// TIA Portal V20 export
TYPE "LBP_typeTMSpindleMT"
TITLE = Tool management / Gestion des outils
// User data type for block LBP_TMSpindleMT [DB1072] / Type de données utilisateur pour bloc LBP_TMSpindleMT [DB1072]
   STRUCT
      MTIF : Array[1..16] of Struct
         DistanceCoding : Int;   // Type of distance coding ($TC_MTP_KD) / Type de codage de distance ($TC_MTP_KD)
         Places : Int;   // Number of locations of the multitool / Nombre d'emplacements Multitool
         Distance : Real;   // Multitool location distance / Distance de l'emplacement Multitool
         NewMTNo : Int;   // MT number of new tool / Numéro MT du nouvel outil
         NewPlace : Int;   // Multitool place number / Numéro d'emplacement Multitool
         OldMTNo : Int;   // MT number of previous tool / Numéro MT de l'outil précédent
         OldPlace : Int;   // Multitool place number / Numéro d'emplacement Multitool
         LocType : Int;   // Tool new: location type / Nouvel outil : type d'emplacement
         SLeft : Int;   // Tool new: size left / Nouvel outil : taille côté gauche
         SRight : Int;   // Tool new: size right / Nouvel outil : taille côté droit
         STop : Int;   // Tool new: size top / Nouvel outil : taille dessus
         SBottom : Int;   // Tool new: size bottom / Nouvel outil : taille dessous
         TInBuffer : Bool;   // ID for tools in buffer / ID pour outils dans tampon
         IgnoreDisabled : Bool;   // Ignore disabled / Ignorer désactivation
         Unload : Bool;   // To be unloaded / À décharger
         Load : Bool;   // To be loaded / À charger
         MasterTool : Bool;   // Tool is the master tool / L'outil est un outil principal
         n26_5 : Bool;   // Reserved / Réservé
         n26_6 : Bool;   // Reserved / Réservé
         HandTool : Bool;   // Hand tool / Outil manuel
         Active : Bool;   // Active tool / Outil actif
         Enabled : Bool;   // Tool enabled / Outil activé
         Disabled : Bool;   // Tool disabled / Outil désactivé
         Measured : Bool;   // Tool measured / Outil mesuré
         Prewarn : Bool;   // Prewarning limit reached / Seuil de préavis atteint
         Change : Bool;   // Tool being changed / Outil en cours de changement
         FixedLoc : Bool;   // Tool fixed location coded / Emplacement fixe d'outil codé
         Used : Bool;   // Tool was in use / Outil a été utilisé
         TNo : Int;   // Tool new: T number / Nouvel outil : numéro d'outil
         Toolholder : Int;   // Toolholder number as tool compensation reference / Numéro de porte-outil en tant que référence pour la compensation d'outil
         MyMag : Int;   // Multitool number the tool is loaded onto / Numéro Multitool dans lequel l'outil est chargé
         MyPlace : Int;   // Multitool place number / Numéro d'emplacement Multitool
         reserved : Array[1..7] of Int;   // Reserved / Réservé
      END_STRUCT;
   END_STRUCT;
   // // MTIF[2].DistanceCoding : Type of distance coding ($TC_MTP_KD) / Type de codage de distance ($TC_MTP_KD)
   // // MTIF[3].DistanceCoding : Type of distance coding ($TC_MTP_KD) / Type de codage de distance ($TC_MTP_KD)
   // // MTIF[4].DistanceCoding : Type of distance coding ($TC_MTP_KD) / Type de codage de distance ($TC_MTP_KD)
   // // MTIF[5].DistanceCoding : Type of distance coding ($TC_MTP_KD) / Type de codage de distance ($TC_MTP_KD)
   // // MTIF[6].DistanceCoding : Type of distance coding ($TC_MTP_KD) / Type de codage de distance ($TC_MTP_KD)
   // // MTIF[7].DistanceCoding : Type of distance coding ($TC_MTP_KD) / Type de codage de distance ($TC_MTP_KD)
   // // MTIF[8].DistanceCoding : Type of distance coding ($TC_MTP_KD) / Type de codage de distance ($TC_MTP_KD)
   // // MTIF[9].DistanceCoding : Type of distance coding ($TC_MTP_KD) / Type de codage de distance ($TC_MTP_KD)
   // // MTIF[10].DistanceCoding : Type of distance coding ($TC_MTP_KD) / Type de codage de distance ($TC_MTP_KD)
   // // MTIF[11].DistanceCoding : Type of distance coding ($TC_MTP_KD) / Type de codage de distance ($TC_MTP_KD)
   // // MTIF[12].DistanceCoding : Type of distance coding ($TC_MTP_KD) / Type de codage de distance ($TC_MTP_KD)
   // // MTIF[13].DistanceCoding : Type of distance coding ($TC_MTP_KD) / Type de codage de distance ($TC_MTP_KD)
   // // MTIF[14].DistanceCoding : Type of distance coding ($TC_MTP_KD) / Type de codage de distance ($TC_MTP_KD)
   // // MTIF[15].DistanceCoding : Type of distance coding ($TC_MTP_KD) / Type de codage de distance ($TC_MTP_KD)
   // // MTIF[16].DistanceCoding : Type of distance coding ($TC_MTP_KD) / Type de codage de distance ($TC_MTP_KD)
   // // MTIF[2].Places : Number of locations of the multitool / Nombre d'emplacements Multitool
   // // MTIF[3].Places : Number of locations of the multitool / Nombre d'emplacements Multitool
   // // MTIF[4].Places : Number of locations of the multitool / Nombre d'emplacements Multitool
   // // MTIF[5].Places : Number of locations of the multitool / Nombre d'emplacements Multitool
   // // MTIF[6].Places : Number of locations of the multitool / Nombre d'emplacements Multitool
   // // MTIF[7].Places : Number of locations of the multitool / Nombre d'emplacements Multitool
   // // MTIF[8].Places : Number of locations of the multitool / Nombre d'emplacements Multitool
   // // MTIF[9].Places : Number of locations of the multitool / Nombre d'emplacements Multitool
   // // MTIF[10].Places : Number of locations of the multitool / Nombre d'emplacements Multitool
   // // MTIF[11].Places : Number of locations of the multitool / Nombre d'emplacements Multitool
   // // MTIF[12].Places : Number of locations of the multitool / Nombre d'emplacements Multitool
   // // MTIF[13].Places : Number of locations of the multitool / Nombre d'emplacements Multitool
   // // MTIF[14].Places : Number of locations of the multitool / Nombre d'emplacements Multitool
   // // MTIF[15].Places : Number of locations of the multitool / Nombre d'emplacements Multitool
   // // MTIF[16].Places : Number of locations of the multitool / Nombre d'emplacements Multitool
   // // MTIF[2].Distance : Multitool location distance / Distance de l'emplacement Multitool
   // // MTIF[3].Distance : Multitool location distance / Distance de l'emplacement Multitool
   // // MTIF[4].Distance : Multitool location distance / Distance de l'emplacement Multitool
   // // MTIF[5].Distance : Multitool location distance / Distance de l'emplacement Multitool
   // // MTIF[6].Distance : Multitool location distance / Distance de l'emplacement Multitool
   // // MTIF[7].Distance : Multitool location distance / Distance de l'emplacement Multitool
   // // MTIF[8].Distance : Multitool location distance / Distance de l'emplacement Multitool
   // // MTIF[9].Distance : Multitool location distance / Distance de l'emplacement Multitool
   // // MTIF[10].Distance : Multitool location distance / Distance de l'emplacement Multitool
   // // MTIF[11].Distance : Multitool location distance / Distance de l'emplacement Multitool
   // // MTIF[12].Distance : Multitool location distance / Distance de l'emplacement Multitool
   // // MTIF[13].Distance : Multitool location distance / Distance de l'emplacement Multitool
   // // MTIF[14].Distance : Multitool location distance / Distance de l'emplacement Multitool
   // // MTIF[15].Distance : Multitool location distance / Distance de l'emplacement Multitool
   // // MTIF[16].Distance : Multitool location distance / Distance de l'emplacement Multitool
   // // MTIF[2].NewMTNo : MT number of new tool / Numéro MT du nouvel outil
   // // MTIF[3].NewMTNo : MT number of new tool / Numéro MT du nouvel outil
   // // MTIF[4].NewMTNo : MT number of new tool / Numéro MT du nouvel outil
   // // MTIF[5].NewMTNo : MT number of new tool / Numéro MT du nouvel outil
   // // MTIF[6].NewMTNo : MT number of new tool / Numéro MT du nouvel outil
   // // MTIF[7].NewMTNo : MT number of new tool / Numéro MT du nouvel outil
   // // MTIF[8].NewMTNo : MT number of new tool / Numéro MT du nouvel outil
   // // MTIF[9].NewMTNo : MT number of new tool / Numéro MT du nouvel outil
   // // MTIF[10].NewMTNo : MT number of new tool / Numéro MT du nouvel outil
   // // MTIF[11].NewMTNo : MT number of new tool / Numéro MT du nouvel outil
   // // MTIF[12].NewMTNo : MT number of new tool / Numéro MT du nouvel outil
   // // MTIF[13].NewMTNo : MT number of new tool / Numéro MT du nouvel outil
   // // MTIF[14].NewMTNo : MT number of new tool / Numéro MT du nouvel outil
   // // MTIF[15].NewMTNo : MT number of new tool / Numéro MT du nouvel outil
   // // MTIF[16].NewMTNo : MT number of new tool / Numéro MT du nouvel outil
   // // MTIF[2].NewPlace : Multitool place number / Numéro d'emplacement Multitool
   // // MTIF[3].NewPlace : Multitool place number / Numéro d'emplacement Multitool
   // // MTIF[4].NewPlace : Multitool place number / Numéro d'emplacement Multitool
   // // MTIF[5].NewPlace : Multitool place number / Numéro d'emplacement Multitool
   // // MTIF[6].NewPlace : Multitool place number / Numéro d'emplacement Multitool
   // // MTIF[7].NewPlace : Multitool place number / Numéro d'emplacement Multitool
   // // MTIF[8].NewPlace : Multitool place number / Numéro d'emplacement Multitool
   // // MTIF[9].NewPlace : Multitool place number / Numéro d'emplacement Multitool
   // // MTIF[10].NewPlace : Multitool place number / Numéro d'emplacement Multitool
   // // MTIF[11].NewPlace : Multitool place number / Numéro d'emplacement Multitool
   // // MTIF[12].NewPlace : Multitool place number / Numéro d'emplacement Multitool
   // // MTIF[13].NewPlace : Multitool place number / Numéro d'emplacement Multitool
   // // MTIF[14].NewPlace : Multitool place number / Numéro d'emplacement Multitool
   // // MTIF[15].NewPlace : Multitool place number / Numéro d'emplacement Multitool
   // // MTIF[16].NewPlace : Multitool place number / Numéro d'emplacement Multitool
   // // MTIF[2].OldMTNo : MT number of previous tool / Numéro MT de l'outil précédent
   // // MTIF[3].OldMTNo : MT number of previous tool / Numéro MT de l'outil précédent
   // // MTIF[4].OldMTNo : MT number of previous tool / Numéro MT de l'outil précédent
   // // MTIF[5].OldMTNo : MT number of previous tool / Numéro MT de l'outil précédent
   // // MTIF[6].OldMTNo : MT number of previous tool / Numéro MT de l'outil précédent
   // // MTIF[7].OldMTNo : MT number of previous tool / Numéro MT de l'outil précédent
   // // MTIF[8].OldMTNo : MT number of previous tool / Numéro MT de l'outil précédent
   // // MTIF[9].OldMTNo : MT number of previous tool / Numéro MT de l'outil précédent
   // // MTIF[10].OldMTNo : MT number of previous tool / Numéro MT de l'outil précédent
   // // MTIF[11].OldMTNo : MT number of previous tool / Numéro MT de l'outil précédent
   // // MTIF[12].OldMTNo : MT number of previous tool / Numéro MT de l'outil précédent
   // // MTIF[13].OldMTNo : MT number of previous tool / Numéro MT de l'outil précédent
   // // MTIF[14].OldMTNo : MT number of previous tool / Numéro MT de l'outil précédent
   // // MTIF[15].OldMTNo : MT number of previous tool / Numéro MT de l'outil précédent
   // // MTIF[16].OldMTNo : MT number of previous tool / Numéro MT de l'outil précédent
   // // MTIF[2].OldPlace : Multitool place number / Numéro d'emplacement Multitool
   // // MTIF[3].OldPlace : Multitool place number / Numéro d'emplacement Multitool
   // // MTIF[4].OldPlace : Multitool place number / Numéro d'emplacement Multitool
   // // MTIF[5].OldPlace : Multitool place number / Numéro d'emplacement Multitool
   // // MTIF[6].OldPlace : Multitool place number / Numéro d'emplacement Multitool
   // // MTIF[7].OldPlace : Multitool place number / Numéro d'emplacement Multitool
   // // MTIF[8].OldPlace : Multitool place number / Numéro d'emplacement Multitool
   // // MTIF[9].OldPlace : Multitool place number / Numéro d'emplacement Multitool
   // // MTIF[10].OldPlace : Multitool place number / Numéro d'emplacement Multitool
   // // MTIF[11].OldPlace : Multitool place number / Numéro d'emplacement Multitool
   // // MTIF[12].OldPlace : Multitool place number / Numéro d'emplacement Multitool
   // // MTIF[13].OldPlace : Multitool place number / Numéro d'emplacement Multitool
   // // MTIF[14].OldPlace : Multitool place number / Numéro d'emplacement Multitool
   // // MTIF[15].OldPlace : Multitool place number / Numéro d'emplacement Multitool
   // // MTIF[16].OldPlace : Multitool place number / Numéro d'emplacement Multitool
   // // MTIF[2].LocType : Tool new: location type / Nouvel outil : type d'emplacement
   // // MTIF[3].LocType : Tool new: location type / Nouvel outil : type d'emplacement
   // // MTIF[4].LocType : Tool new: location type / Nouvel outil : type d'emplacement
   // // MTIF[5].LocType : Tool new: location type / Nouvel outil : type d'emplacement
   // // MTIF[6].LocType : Tool new: location type / Nouvel outil : type d'emplacement
   // // MTIF[7].LocType : Tool new: location type / Nouvel outil : type d'emplacement
   // // MTIF[8].LocType : Tool new: location type / Nouvel outil : type d'emplacement
   // // MTIF[9].LocType : Tool new: location type / Nouvel outil : type d'emplacement
   // // MTIF[10].LocType : Tool new: location type / Nouvel outil : type d'emplacement
   // // MTIF[11].LocType : Tool new: location type / Nouvel outil : type d'emplacement
   // // MTIF[12].LocType : Tool new: location type / Nouvel outil : type d'emplacement
   // // MTIF[13].LocType : Tool new: location type / Nouvel outil : type d'emplacement
   // // MTIF[14].LocType : Tool new: location type / Nouvel outil : type d'emplacement
   // // MTIF[15].LocType : Tool new: location type / Nouvel outil : type d'emplacement
   // // MTIF[16].LocType : Tool new: location type / Nouvel outil : type d'emplacement
   // // MTIF[2].SLeft : Tool new: size left / Nouvel outil : taille côté gauche
   // // MTIF[3].SLeft : Tool new: size left / Nouvel outil : taille côté gauche
   // // MTIF[4].SLeft : Tool new: size left / Nouvel outil : taille côté gauche
   // // MTIF[5].SLeft : Tool new: size left / Nouvel outil : taille côté gauche
   // // MTIF[6].SLeft : Tool new: size left / Nouvel outil : taille côté gauche
   // // MTIF[7].SLeft : Tool new: size left / Nouvel outil : taille côté gauche
   // // MTIF[8].SLeft : Tool new: size left / Nouvel outil : taille côté gauche
   // // MTIF[9].SLeft : Tool new: size left / Nouvel outil : taille côté gauche
   // // MTIF[10].SLeft : Tool new: size left / Nouvel outil : taille côté gauche
   // // MTIF[11].SLeft : Tool new: size left / Nouvel outil : taille côté gauche
   // // MTIF[12].SLeft : Tool new: size left / Nouvel outil : taille côté gauche
   // // MTIF[13].SLeft : Tool new: size left / Nouvel outil : taille côté gauche
   // // MTIF[14].SLeft : Tool new: size left / Nouvel outil : taille côté gauche
   // // MTIF[15].SLeft : Tool new: size left / Nouvel outil : taille côté gauche
   // // MTIF[16].SLeft : Tool new: size left / Nouvel outil : taille côté gauche
   // // MTIF[2].SRight : Tool new: size right / Nouvel outil : taille côté droit
   // // MTIF[3].SRight : Tool new: size right / Nouvel outil : taille côté droit
   // // MTIF[4].SRight : Tool new: size right / Nouvel outil : taille côté droit
   // // MTIF[5].SRight : Tool new: size right / Nouvel outil : taille côté droit
   // // MTIF[6].SRight : Tool new: size right / Nouvel outil : taille côté droit
   // // MTIF[7].SRight : Tool new: size right / Nouvel outil : taille côté droit
   // // MTIF[8].SRight : Tool new: size right / Nouvel outil : taille côté droit
   // // MTIF[9].SRight : Tool new: size right / Nouvel outil : taille côté droit
   // // MTIF[10].SRight : Tool new: size right / Nouvel outil : taille côté droit
   // // MTIF[11].SRight : Tool new: size right / Nouvel outil : taille côté droit
   // // MTIF[12].SRight : Tool new: size right / Nouvel outil : taille côté droit
   // // MTIF[13].SRight : Tool new: size right / Nouvel outil : taille côté droit
   // // MTIF[14].SRight : Tool new: size right / Nouvel outil : taille côté droit
   // // MTIF[15].SRight : Tool new: size right / Nouvel outil : taille côté droit
   // // MTIF[16].SRight : Tool new: size right / Nouvel outil : taille côté droit
   // // MTIF[2].STop : Tool new: size top / Nouvel outil : taille dessus
   // // MTIF[3].STop : Tool new: size top / Nouvel outil : taille dessus
   // // MTIF[4].STop : Tool new: size top / Nouvel outil : taille dessus
   // // MTIF[5].STop : Tool new: size top / Nouvel outil : taille dessus
   // // MTIF[6].STop : Tool new: size top / Nouvel outil : taille dessus
   // // MTIF[7].STop : Tool new: size top / Nouvel outil : taille dessus
   // // MTIF[8].STop : Tool new: size top / Nouvel outil : taille dessus
   // // MTIF[9].STop : Tool new: size top / Nouvel outil : taille dessus
   // // MTIF[10].STop : Tool new: size top / Nouvel outil : taille dessus
   // // MTIF[11].STop : Tool new: size top / Nouvel outil : taille dessus
   // // MTIF[12].STop : Tool new: size top / Nouvel outil : taille dessus
   // // MTIF[13].STop : Tool new: size top / Nouvel outil : taille dessus
   // // MTIF[14].STop : Tool new: size top / Nouvel outil : taille dessus
   // // MTIF[15].STop : Tool new: size top / Nouvel outil : taille dessus
   // // MTIF[16].STop : Tool new: size top / Nouvel outil : taille dessus
   // // MTIF[2].SBottom : Tool new: size bottom / Nouvel outil : taille dessous
   // // MTIF[3].SBottom : Tool new: size bottom / Nouvel outil : taille dessous
   // // MTIF[4].SBottom : Tool new: size bottom / Nouvel outil : taille dessous
   // // MTIF[5].SBottom : Tool new: size bottom / Nouvel outil : taille dessous
   // // MTIF[6].SBottom : Tool new: size bottom / Nouvel outil : taille dessous
   // // MTIF[7].SBottom : Tool new: size bottom / Nouvel outil : taille dessous
   // // MTIF[8].SBottom : Tool new: size bottom / Nouvel outil : taille dessous
   // // MTIF[9].SBottom : Tool new: size bottom / Nouvel outil : taille dessous
   // // MTIF[10].SBottom : Tool new: size bottom / Nouvel outil : taille dessous
   // // MTIF[11].SBottom : Tool new: size bottom / Nouvel outil : taille dessous
   // // MTIF[12].SBottom : Tool new: size bottom / Nouvel outil : taille dessous
   // // MTIF[13].SBottom : Tool new: size bottom / Nouvel outil : taille dessous
   // // MTIF[14].SBottom : Tool new: size bottom / Nouvel outil : taille dessous
   // // MTIF[15].SBottom : Tool new: size bottom / Nouvel outil : taille dessous
   // // MTIF[16].SBottom : Tool new: size bottom / Nouvel outil : taille dessous
   // // MTIF[2].TInBuffer : ID for tools in buffer / ID pour outils dans tampon
   // // MTIF[3].TInBuffer : ID for tools in buffer / ID pour outils dans tampon
   // // MTIF[4].TInBuffer : ID for tools in buffer / ID pour outils dans tampon
   // // MTIF[5].TInBuffer : ID for tools in buffer / ID pour outils dans tampon
   // // MTIF[6].TInBuffer : ID for tools in buffer / ID pour outils dans tampon
   // // MTIF[7].TInBuffer : ID for tools in buffer / ID pour outils dans tampon
   // // MTIF[8].TInBuffer : ID for tools in buffer / ID pour outils dans tampon
   // // MTIF[9].TInBuffer : ID for tools in buffer / ID pour outils dans tampon
   // // MTIF[10].TInBuffer : ID for tools in buffer / ID pour outils dans tampon
   // // MTIF[11].TInBuffer : ID for tools in buffer / ID pour outils dans tampon
   // // MTIF[12].TInBuffer : ID for tools in buffer / ID pour outils dans tampon
   // // MTIF[13].TInBuffer : ID for tools in buffer / ID pour outils dans tampon
   // // MTIF[14].TInBuffer : ID for tools in buffer / ID pour outils dans tampon
   // // MTIF[15].TInBuffer : ID for tools in buffer / ID pour outils dans tampon
   // // MTIF[16].TInBuffer : ID for tools in buffer / ID pour outils dans tampon
   // // MTIF[2].IgnoreDisabled : Ignore disabled / Ignorer désactivation
   // // MTIF[3].IgnoreDisabled : Ignore disabled / Ignorer désactivation
   // // MTIF[4].IgnoreDisabled : Ignore disabled / Ignorer désactivation
   // // MTIF[5].IgnoreDisabled : Ignore disabled / Ignorer désactivation
   // // MTIF[6].IgnoreDisabled : Ignore disabled / Ignorer désactivation
   // // MTIF[7].IgnoreDisabled : Ignore disabled / Ignorer désactivation
   // // MTIF[8].IgnoreDisabled : Ignore disabled / Ignorer désactivation
   // // MTIF[9].IgnoreDisabled : Ignore disabled / Ignorer désactivation
   // // MTIF[10].IgnoreDisabled : Ignore disabled / Ignorer désactivation
   // // MTIF[11].IgnoreDisabled : Ignore disabled / Ignorer désactivation
   // // MTIF[12].IgnoreDisabled : Ignore disabled / Ignorer désactivation
   // // MTIF[13].IgnoreDisabled : Ignore disabled / Ignorer désactivation
   // // MTIF[14].IgnoreDisabled : Ignore disabled / Ignorer désactivation
   // // MTIF[15].IgnoreDisabled : Ignore disabled / Ignorer désactivation
   // // MTIF[16].IgnoreDisabled : Ignore disabled / Ignorer désactivation
   // // MTIF[2].Unload : To be unloaded / À décharger
   // // MTIF[3].Unload : To be unloaded / À décharger
   // // MTIF[4].Unload : To be unloaded / À décharger
   // // MTIF[5].Unload : To be unloaded / À décharger
   // // MTIF[6].Unload : To be unloaded / À décharger
   // // MTIF[7].Unload : To be unloaded / À décharger
   // // MTIF[8].Unload : To be unloaded / À décharger
   // // MTIF[9].Unload : To be unloaded / À décharger
   // // MTIF[10].Unload : To be unloaded / À décharger
   // // MTIF[11].Unload : To be unloaded / À décharger
   // // MTIF[12].Unload : To be unloaded / À décharger
   // // MTIF[13].Unload : To be unloaded / À décharger
   // // MTIF[14].Unload : To be unloaded / À décharger
   // // MTIF[15].Unload : To be unloaded / À décharger
   // // MTIF[16].Unload : To be unloaded / À décharger
   // // MTIF[2].Load : To be loaded / À charger
   // // MTIF[3].Load : To be loaded / À charger
   // // MTIF[4].Load : To be loaded / À charger
   // // MTIF[5].Load : To be loaded / À charger
   // // MTIF[6].Load : To be loaded / À charger
   // // MTIF[7].Load : To be loaded / À charger
   // // MTIF[8].Load : To be loaded / À charger
   // // MTIF[9].Load : To be loaded / À charger
   // // MTIF[10].Load : To be loaded / À charger
   // // MTIF[11].Load : To be loaded / À charger
   // // MTIF[12].Load : To be loaded / À charger
   // // MTIF[13].Load : To be loaded / À charger
   // // MTIF[14].Load : To be loaded / À charger
   // // MTIF[15].Load : To be loaded / À charger
   // // MTIF[16].Load : To be loaded / À charger
   // // MTIF[2].MasterTool : Tool is the master tool / L'outil est un outil principal
   // // MTIF[3].MasterTool : Tool is the master tool / L'outil est un outil principal
   // // MTIF[4].MasterTool : Tool is the master tool / L'outil est un outil principal
   // // MTIF[5].MasterTool : Tool is the master tool / L'outil est un outil principal
   // // MTIF[6].MasterTool : Tool is the master tool / L'outil est un outil principal
   // // MTIF[7].MasterTool : Tool is the master tool / L'outil est un outil principal
   // // MTIF[8].MasterTool : Tool is the master tool / L'outil est un outil principal
   // // MTIF[9].MasterTool : Tool is the master tool / L'outil est un outil principal
   // // MTIF[10].MasterTool : Tool is the master tool / L'outil est un outil principal
   // // MTIF[11].MasterTool : Tool is the master tool / L'outil est un outil principal
   // // MTIF[12].MasterTool : Tool is the master tool / L'outil est un outil principal
   // // MTIF[13].MasterTool : Tool is the master tool / L'outil est un outil principal
   // // MTIF[14].MasterTool : Tool is the master tool / L'outil est un outil principal
   // // MTIF[15].MasterTool : Tool is the master tool / L'outil est un outil principal
   // // MTIF[16].MasterTool : Tool is the master tool / L'outil est un outil principal
   // // MTIF[2].n26_5 : Reserved / Réservé
   // // MTIF[3].n26_5 : Reserved / Réservé
   // // MTIF[4].n26_5 : Reserved / Réservé
   // // MTIF[5].n26_5 : Reserved / Réservé
   // // MTIF[6].n26_5 : Reserved / Réservé
   // // MTIF[7].n26_5 : Reserved / Réservé
   // // MTIF[8].n26_5 : Reserved / Réservé
   // // MTIF[9].n26_5 : Reserved / Réservé
   // // MTIF[10].n26_5 : Reserved / Réservé
   // // MTIF[11].n26_5 : Reserved / Réservé
   // // MTIF[12].n26_5 : Reserved / Réservé
   // // MTIF[13].n26_5 : Reserved / Réservé
   // // MTIF[14].n26_5 : Reserved / Réservé
   // // MTIF[15].n26_5 : Reserved / Réservé
   // // MTIF[16].n26_5 : Reserved / Réservé
   // // MTIF[2].n26_6 : Reserved / Réservé
   // // MTIF[3].n26_6 : Reserved / Réservé
   // // MTIF[4].n26_6 : Reserved / Réservé
   // // MTIF[5].n26_6 : Reserved / Réservé
   // // MTIF[6].n26_6 : Reserved / Réservé
   // // MTIF[7].n26_6 : Reserved / Réservé
   // // MTIF[8].n26_6 : Reserved / Réservé
   // // MTIF[9].n26_6 : Reserved / Réservé
   // // MTIF[10].n26_6 : Reserved / Réservé
   // // MTIF[11].n26_6 : Reserved / Réservé
   // // MTIF[12].n26_6 : Reserved / Réservé
   // // MTIF[13].n26_6 : Reserved / Réservé
   // // MTIF[14].n26_6 : Reserved / Réservé
   // // MTIF[15].n26_6 : Reserved / Réservé
   // // MTIF[16].n26_6 : Reserved / Réservé
   // // MTIF[2].HandTool : Hand tool / Outil manuel
   // // MTIF[3].HandTool : Hand tool / Outil manuel
   // // MTIF[4].HandTool : Hand tool / Outil manuel
   // // MTIF[5].HandTool : Hand tool / Outil manuel
   // // MTIF[6].HandTool : Hand tool / Outil manuel
   // // MTIF[7].HandTool : Hand tool / Outil manuel
   // // MTIF[8].HandTool : Hand tool / Outil manuel
   // // MTIF[9].HandTool : Hand tool / Outil manuel
   // // MTIF[10].HandTool : Hand tool / Outil manuel
   // // MTIF[11].HandTool : Hand tool / Outil manuel
   // // MTIF[12].HandTool : Hand tool / Outil manuel
   // // MTIF[13].HandTool : Hand tool / Outil manuel
   // // MTIF[14].HandTool : Hand tool / Outil manuel
   // // MTIF[15].HandTool : Hand tool / Outil manuel
   // // MTIF[16].HandTool : Hand tool / Outil manuel
   // // MTIF[2].Active : Active tool / Outil actif
   // // MTIF[3].Active : Active tool / Outil actif
   // // MTIF[4].Active : Active tool / Outil actif
   // // MTIF[5].Active : Active tool / Outil actif
   // // MTIF[6].Active : Active tool / Outil actif
   // // MTIF[7].Active : Active tool / Outil actif
   // // MTIF[8].Active : Active tool / Outil actif
   // // MTIF[9].Active : Active tool / Outil actif
   // // MTIF[10].Active : Active tool / Outil actif
   // // MTIF[11].Active : Active tool / Outil actif
   // // MTIF[12].Active : Active tool / Outil actif
   // // MTIF[13].Active : Active tool / Outil actif
   // // MTIF[14].Active : Active tool / Outil actif
   // // MTIF[15].Active : Active tool / Outil actif
   // // MTIF[16].Active : Active tool / Outil actif
   // // MTIF[2].Enabled : Tool enabled / Outil activé
   // // MTIF[3].Enabled : Tool enabled / Outil activé
   // // MTIF[4].Enabled : Tool enabled / Outil activé
   // // MTIF[5].Enabled : Tool enabled / Outil activé
   // // MTIF[6].Enabled : Tool enabled / Outil activé
   // // MTIF[7].Enabled : Tool enabled / Outil activé
   // // MTIF[8].Enabled : Tool enabled / Outil activé
   // // MTIF[9].Enabled : Tool enabled / Outil activé
   // // MTIF[10].Enabled : Tool enabled / Outil activé
   // // MTIF[11].Enabled : Tool enabled / Outil activé
   // // MTIF[12].Enabled : Tool enabled / Outil activé
   // // MTIF[13].Enabled : Tool enabled / Outil activé
   // // MTIF[14].Enabled : Tool enabled / Outil activé
   // // MTIF[15].Enabled : Tool enabled / Outil activé
   // // MTIF[16].Enabled : Tool enabled / Outil activé
   // // MTIF[2].Disabled : Tool disabled / Outil désactivé
   // // MTIF[3].Disabled : Tool disabled / Outil désactivé
   // // MTIF[4].Disabled : Tool disabled / Outil désactivé
   // // MTIF[5].Disabled : Tool disabled / Outil désactivé
   // // MTIF[6].Disabled : Tool disabled / Outil désactivé
   // // MTIF[7].Disabled : Tool disabled / Outil désactivé
   // // MTIF[8].Disabled : Tool disabled / Outil désactivé
   // // MTIF[9].Disabled : Tool disabled / Outil désactivé
   // // MTIF[10].Disabled : Tool disabled / Outil désactivé
   // // MTIF[11].Disabled : Tool disabled / Outil désactivé
   // // MTIF[12].Disabled : Tool disabled / Outil désactivé
   // // MTIF[13].Disabled : Tool disabled / Outil désactivé
   // // MTIF[14].Disabled : Tool disabled / Outil désactivé
   // // MTIF[15].Disabled : Tool disabled / Outil désactivé
   // // MTIF[16].Disabled : Tool disabled / Outil désactivé
   // // MTIF[2].Measured : Tool measured / Outil mesuré
   // // MTIF[3].Measured : Tool measured / Outil mesuré
   // // MTIF[4].Measured : Tool measured / Outil mesuré
   // // MTIF[5].Measured : Tool measured / Outil mesuré
   // // MTIF[6].Measured : Tool measured / Outil mesuré
   // // MTIF[7].Measured : Tool measured / Outil mesuré
   // // MTIF[8].Measured : Tool measured / Outil mesuré
   // // MTIF[9].Measured : Tool measured / Outil mesuré
   // // MTIF[10].Measured : Tool measured / Outil mesuré
   // // MTIF[11].Measured : Tool measured / Outil mesuré
   // // MTIF[12].Measured : Tool measured / Outil mesuré
   // // MTIF[13].Measured : Tool measured / Outil mesuré
   // // MTIF[14].Measured : Tool measured / Outil mesuré
   // // MTIF[15].Measured : Tool measured / Outil mesuré
   // // MTIF[16].Measured : Tool measured / Outil mesuré
   // // MTIF[2].Prewarn : Prewarning limit reached / Seuil de préavis atteint
   // // MTIF[3].Prewarn : Prewarning limit reached / Seuil de préavis atteint
   // // MTIF[4].Prewarn : Prewarning limit reached / Seuil de préavis atteint
   // // MTIF[5].Prewarn : Prewarning limit reached / Seuil de préavis atteint
   // // MTIF[6].Prewarn : Prewarning limit reached / Seuil de préavis atteint
   // // MTIF[7].Prewarn : Prewarning limit reached / Seuil de préavis atteint
   // // MTIF[8].Prewarn : Prewarning limit reached / Seuil de préavis atteint
   // // MTIF[9].Prewarn : Prewarning limit reached / Seuil de préavis atteint
   // // MTIF[10].Prewarn : Prewarning limit reached / Seuil de préavis atteint
   // // MTIF[11].Prewarn : Prewarning limit reached / Seuil de préavis atteint
   // // MTIF[12].Prewarn : Prewarning limit reached / Seuil de préavis atteint
   // // MTIF[13].Prewarn : Prewarning limit reached / Seuil de préavis atteint
   // // MTIF[14].Prewarn : Prewarning limit reached / Seuil de préavis atteint
   // // MTIF[15].Prewarn : Prewarning limit reached / Seuil de préavis atteint
   // // MTIF[16].Prewarn : Prewarning limit reached / Seuil de préavis atteint
   // // MTIF[2].Change : Tool being changed / Outil en cours de changement
   // // MTIF[3].Change : Tool being changed / Outil en cours de changement
   // // MTIF[4].Change : Tool being changed / Outil en cours de changement
   // // MTIF[5].Change : Tool being changed / Outil en cours de changement
   // // MTIF[6].Change : Tool being changed / Outil en cours de changement
   // // MTIF[7].Change : Tool being changed / Outil en cours de changement
   // // MTIF[8].Change : Tool being changed / Outil en cours de changement
   // // MTIF[9].Change : Tool being changed / Outil en cours de changement
   // // MTIF[10].Change : Tool being changed / Outil en cours de changement
   // // MTIF[11].Change : Tool being changed / Outil en cours de changement
   // // MTIF[12].Change : Tool being changed / Outil en cours de changement
   // // MTIF[13].Change : Tool being changed / Outil en cours de changement
   // // MTIF[14].Change : Tool being changed / Outil en cours de changement
   // // MTIF[15].Change : Tool being changed / Outil en cours de changement
   // // MTIF[16].Change : Tool being changed / Outil en cours de changement
   // // MTIF[2].FixedLoc : Tool fixed location coded / Emplacement fixe d'outil codé
   // // MTIF[3].FixedLoc : Tool fixed location coded / Emplacement fixe d'outil codé
   // // MTIF[4].FixedLoc : Tool fixed location coded / Emplacement fixe d'outil codé
   // // MTIF[5].FixedLoc : Tool fixed location coded / Emplacement fixe d'outil codé
   // // MTIF[6].FixedLoc : Tool fixed location coded / Emplacement fixe d'outil codé
   // // MTIF[7].FixedLoc : Tool fixed location coded / Emplacement fixe d'outil codé
   // // MTIF[8].FixedLoc : Tool fixed location coded / Emplacement fixe d'outil codé
   // // MTIF[9].FixedLoc : Tool fixed location coded / Emplacement fixe d'outil codé
   // // MTIF[10].FixedLoc : Tool fixed location coded / Emplacement fixe d'outil codé
   // // MTIF[11].FixedLoc : Tool fixed location coded / Emplacement fixe d'outil codé
   // // MTIF[12].FixedLoc : Tool fixed location coded / Emplacement fixe d'outil codé
   // // MTIF[13].FixedLoc : Tool fixed location coded / Emplacement fixe d'outil codé
   // // MTIF[14].FixedLoc : Tool fixed location coded / Emplacement fixe d'outil codé
   // // MTIF[15].FixedLoc : Tool fixed location coded / Emplacement fixe d'outil codé
   // // MTIF[16].FixedLoc : Tool fixed location coded / Emplacement fixe d'outil codé
   // // MTIF[2].Used : Tool was in use / Outil a été utilisé
   // // MTIF[3].Used : Tool was in use / Outil a été utilisé
   // // MTIF[4].Used : Tool was in use / Outil a été utilisé
   // // MTIF[5].Used : Tool was in use / Outil a été utilisé
   // // MTIF[6].Used : Tool was in use / Outil a été utilisé
   // // MTIF[7].Used : Tool was in use / Outil a été utilisé
   // // MTIF[8].Used : Tool was in use / Outil a été utilisé
   // // MTIF[9].Used : Tool was in use / Outil a été utilisé
   // // MTIF[10].Used : Tool was in use / Outil a été utilisé
   // // MTIF[11].Used : Tool was in use / Outil a été utilisé
   // // MTIF[12].Used : Tool was in use / Outil a été utilisé
   // // MTIF[13].Used : Tool was in use / Outil a été utilisé
   // // MTIF[14].Used : Tool was in use / Outil a été utilisé
   // // MTIF[15].Used : Tool was in use / Outil a été utilisé
   // // MTIF[16].Used : Tool was in use / Outil a été utilisé
   // // MTIF[2].TNo : Tool new: T number / Nouvel outil : numéro d'outil
   // // MTIF[3].TNo : Tool new: T number / Nouvel outil : numéro d'outil
   // // MTIF[4].TNo : Tool new: T number / Nouvel outil : numéro d'outil
   // // MTIF[5].TNo : Tool new: T number / Nouvel outil : numéro d'outil
   // // MTIF[6].TNo : Tool new: T number / Nouvel outil : numéro d'outil
   // // MTIF[7].TNo : Tool new: T number / Nouvel outil : numéro d'outil
   // // MTIF[8].TNo : Tool new: T number / Nouvel outil : numéro d'outil
   // // MTIF[9].TNo : Tool new: T number / Nouvel outil : numéro d'outil
   // // MTIF[10].TNo : Tool new: T number / Nouvel outil : numéro d'outil
   // // MTIF[11].TNo : Tool new: T number / Nouvel outil : numéro d'outil
   // // MTIF[12].TNo : Tool new: T number / Nouvel outil : numéro d'outil
   // // MTIF[13].TNo : Tool new: T number / Nouvel outil : numéro d'outil
   // // MTIF[14].TNo : Tool new: T number / Nouvel outil : numéro d'outil
   // // MTIF[15].TNo : Tool new: T number / Nouvel outil : numéro d'outil
   // // MTIF[16].TNo : Tool new: T number / Nouvel outil : numéro d'outil
   // // MTIF[2].Toolholder : Toolholder number as tool compensation reference / Numéro de porte-outil en tant que référence pour la compensation d'outil
   // // MTIF[3].Toolholder : Toolholder number as tool compensation reference / Numéro de porte-outil en tant que référence pour la compensation d'outil
   // // MTIF[4].Toolholder : Toolholder number as tool compensation reference / Numéro de porte-outil en tant que référence pour la compensation d'outil
   // // MTIF[5].Toolholder : Toolholder number as tool compensation reference / Numéro de porte-outil en tant que référence pour la compensation d'outil
   // // MTIF[6].Toolholder : Toolholder number as tool compensation reference / Numéro de porte-outil en tant que référence pour la compensation d'outil
   // // MTIF[7].Toolholder : Toolholder number as tool compensation reference / Numéro de porte-outil en tant que référence pour la compensation d'outil
   // // MTIF[8].Toolholder : Toolholder number as tool compensation reference / Numéro de porte-outil en tant que référence pour la compensation d'outil
   // // MTIF[9].Toolholder : Toolholder number as tool compensation reference / Numéro de porte-outil en tant que référence pour la compensation d'outil
   // // MTIF[10].Toolholder : Toolholder number as tool compensation reference / Numéro de porte-outil en tant que référence pour la compensation d'outil
   // // MTIF[11].Toolholder : Toolholder number as tool compensation reference / Numéro de porte-outil en tant que référence pour la compensation d'outil
   // // MTIF[12].Toolholder : Toolholder number as tool compensation reference / Numéro de porte-outil en tant que référence pour la compensation d'outil
   // // MTIF[13].Toolholder : Toolholder number as tool compensation reference / Numéro de porte-outil en tant que référence pour la compensation d'outil
   // // MTIF[14].Toolholder : Toolholder number as tool compensation reference / Numéro de porte-outil en tant que référence pour la compensation d'outil
   // // MTIF[15].Toolholder : Toolholder number as tool compensation reference / Numéro de porte-outil en tant que référence pour la compensation d'outil
   // // MTIF[16].Toolholder : Toolholder number as tool compensation reference / Numéro de porte-outil en tant que référence pour la compensation d'outil
   // // MTIF[2].MyMag : Multitool number the tool is loaded onto / Numéro Multitool dans lequel l'outil est chargé
   // // MTIF[3].MyMag : Multitool number the tool is loaded onto / Numéro Multitool dans lequel l'outil est chargé
   // // MTIF[4].MyMag : Multitool number the tool is loaded onto / Numéro Multitool dans lequel l'outil est chargé
   // // MTIF[5].MyMag : Multitool number the tool is loaded onto / Numéro Multitool dans lequel l'outil est chargé
   // // MTIF[6].MyMag : Multitool number the tool is loaded onto / Numéro Multitool dans lequel l'outil est chargé
   // // MTIF[7].MyMag : Multitool number the tool is loaded onto / Numéro Multitool dans lequel l'outil est chargé
   // // MTIF[8].MyMag : Multitool number the tool is loaded onto / Numéro Multitool dans lequel l'outil est chargé
   // // MTIF[9].MyMag : Multitool number the tool is loaded onto / Numéro Multitool dans lequel l'outil est chargé
   // // MTIF[10].MyMag : Multitool number the tool is loaded onto / Numéro Multitool dans lequel l'outil est chargé
   // // MTIF[11].MyMag : Multitool number the tool is loaded onto / Numéro Multitool dans lequel l'outil est chargé
   // // MTIF[12].MyMag : Multitool number the tool is loaded onto / Numéro Multitool dans lequel l'outil est chargé
   // // MTIF[13].MyMag : Multitool number the tool is loaded onto / Numéro Multitool dans lequel l'outil est chargé
   // // MTIF[14].MyMag : Multitool number the tool is loaded onto / Numéro Multitool dans lequel l'outil est chargé
   // // MTIF[15].MyMag : Multitool number the tool is loaded onto / Numéro Multitool dans lequel l'outil est chargé
   // // MTIF[16].MyMag : Multitool number the tool is loaded onto / Numéro Multitool dans lequel l'outil est chargé
   // // MTIF[2].MyPlace : Multitool place number / Numéro d'emplacement Multitool
   // // MTIF[3].MyPlace : Multitool place number / Numéro d'emplacement Multitool
   // // MTIF[4].MyPlace : Multitool place number / Numéro d'emplacement Multitool
   // // MTIF[5].MyPlace : Multitool place number / Numéro d'emplacement Multitool
   // // MTIF[6].MyPlace : Multitool place number / Numéro d'emplacement Multitool
   // // MTIF[7].MyPlace : Multitool place number / Numéro d'emplacement Multitool
   // // MTIF[8].MyPlace : Multitool place number / Numéro d'emplacement Multitool
   // // MTIF[9].MyPlace : Multitool place number / Numéro d'emplacement Multitool
   // // MTIF[10].MyPlace : Multitool place number / Numéro d'emplacement Multitool
   // // MTIF[11].MyPlace : Multitool place number / Numéro d'emplacement Multitool
   // // MTIF[12].MyPlace : Multitool place number / Numéro d'emplacement Multitool
   // // MTIF[13].MyPlace : Multitool place number / Numéro d'emplacement Multitool
   // // MTIF[14].MyPlace : Multitool place number / Numéro d'emplacement Multitool
   // // MTIF[15].MyPlace : Multitool place number / Numéro d'emplacement Multitool
   // // MTIF[16].MyPlace : Multitool place number / Numéro d'emplacement Multitool
   // // MTIF[2].reserved : Reserved / Réservé
   // // MTIF[3].reserved : Reserved / Réservé
   // // MTIF[4].reserved : Reserved / Réservé
   // // MTIF[5].reserved : Reserved / Réservé
   // // MTIF[6].reserved : Reserved / Réservé
   // // MTIF[7].reserved : Reserved / Réservé
   // // MTIF[8].reserved : Reserved / Réservé
   // // MTIF[9].reserved : Reserved / Réservé
   // // MTIF[10].reserved : Reserved / Réservé
   // // MTIF[11].reserved : Reserved / Réservé
   // // MTIF[12].reserved : Reserved / Réservé
   // // MTIF[13].reserved : Reserved / Réservé
   // // MTIF[14].reserved : Reserved / Réservé
   // // MTIF[15].reserved : Reserved / Réservé
   // // MTIF[16].reserved : Reserved / Réservé
END_TYPE
